TYPE E_SYSTEM_OSType : (
	E_OS_UNKNOWN,
	E_OS_WINCE,
	E_OS_WINDOWS
);

END_TYPE

(* stored: Version 1.1.0.1
   DUT E_SYSTEM_OSType: Id {512c7970-af37-4c3d-ae8b-32758b51bea6} *)
